Fanuc KAREL source: ks00007.KL

PROGRAM KS00007
%STACKSIZE=65535
%PRIORITY=65535
%NOLOCKGROUP
VAR
FLAG : BOOLEAN
N : INTEGER
STATUS : INTEGER
PN : STRING[80]
VN : STRING[80]
-- UNRESOLVED DECLARATIONS (source type spelling not recovered)
-- A : TYPE_0x1100 (type_u16=0x1100)
-- B : TYPE_0x1100 (type_u16=0x1100)
BEGIN
PN=''
VN='A'
-- UNRESOLVED_PC line 19 opcodes [27 22 22 2A 22 2A 22 22 B0] marker_code=27
END KS00007
